FUNCTION_BLOCK C_HTTP_HEADER EXTENDS C_HTTP_BASE
VAR_INPUT
END_VAR
VAR_OUTPUT
END_VAR
VAR
	_FieldName 	: STRING(255);
	_HeaderField: STRING(255);
END_VAR

METHOD Equals : BOOL
VAR_INPUT
	IN_HEADER : POINTER TO C_HTTP_HEADER;
END_VAR
VAR
	_stringInternal 	: STRING(255);
	_stringInput 		: STRING(255);
	_lenString			: INT;
	_i 					: DINT;
END_VAR
IF LEN(IN_HEADER^.Field_Name) <> LEN(THIS^.Field_Name) THEN
	Equals := FALSE;
ELSIF LEN(IN_HEADER^.Header_Field) <> LEN(THIS^.Header_Field) THEN
	Equals := FALSE;
ELSE
	_stringInternal := THIS^.Field_Name;
	_stringInput := IN_HEADER^.Field_Name;
	_lenString := LEN(_stringInternal);
	_i := MEMCMP(ADR(_stringinternal),ADR(_stringInput), _lenString);
	IF _i <> 0 THEN
		Equals := FALSE;
	ELSE
		_stringInternal := THIS^.Header_Field;
		_stringInput := IN_HEADER^.Header_Field;
		_lenString := LEN(_stringInternal);
		_i := MEMCMP(ADR(_stringinternal),ADR(_stringInput), _lenString);
		IF _i <> 0 THEN
			Equals := FALSE;
		ELSE
			Equals := TRUE;
		END_IF
	END_IF
END_IF
END_METHOD

METHOD FB_init : BOOL
VAR_INPUT
	bInitRetains : BOOL; // if TRUE, the retain variables are initialized (warm start / cold start)
	bInCopyCode : BOOL;  // if TRUE, the instance afterwards gets moved into the copy code (online change)
	Name : STRING(255);
END_VAR
_FieldName := Name;
END_METHOD

PROPERTY Field_Name : STRING(255)
GET
Field_Name := _FieldName;
END_GET
SET
_FieldName := Field_Name;
END_SET
END_PROPERTY

PROPERTY Header_Field : STRING(255)
GET
Header_Field := _HeaderField;
END_GET
SET
_HeaderField := Header_Field;
END_SET
END_PROPERTY

METHOD Parse : RETURN_CODE
VAR_INPUT
	IN_STRING	: STRING(255);
END_VAR
VAR 
	_DELIMIT_POSITION : INT;
	_ENDLINE_POSITION : INT;
END_VAR
_DELIMIT_POSITION := FIND(IN_STRING, SUPER^.Header_Delimiter);
IF _DELIMIT_POSITION = 0 THEN
	Parse := ph_lv0.LV0_RETURNCODE.RETURN_ERROR + 1;
ELSE
	_ENDLINE_POSITION := FIND(IN_STRING, SUPER^.Line_Terminator);
	IF _ENDLINE_POSITION = 0 THEN
		Parse := ph_lv0.LV0_RETURNCODE.RETURN_ERROR + 2;
	ELSE
		_FieldName := MID(IN_STRING, _DELIMIT_POSITION - 1, 1);
		_HeaderField := MID(IN_STRING, _ENDLINE_POSITION - (_DELIMIT_POSITION + 2), _DELIMIT_POSITION + 2); 
		Parse := ph_lv0.LV0_RETURNCODE.RETURN_SUCCESS;
	END_IF
END_IF
END_METHOD

METHOD ToString : String(255)
VAR_INPUT
END_VAR
ToString := CONCAT(THIS^.Field_Name,
				CONCAT(SUPER^.Header_Delimiter, 
					CONCAT(THIS^.Header_Field,
						SUPER^.Line_Terminator
					)
				)
			);
END_METHOD

END_FUNCTION_BLOCK

(* stored: Version 1.1.0.1, ProductVersion 3.1.4019.2
   POU C_HTTP_HEADER: Id {f4916d40-e672-4a39-af07-e680b56b31a1}, SpecialFunc None
   Folder Methods: Id {db0984ec-abb7-47f0-9af2-a9a0dd131973}
   Folder Properties: Id {f10153ac-78e0-47cd-a140-91303f7d4cce}
   Method Equals: Id {3902d8e9-12a8-4da2-98b3-710cc8dffbd1}
   Method FB_init: Id {8a629b36-7f23-4909-b667-670fcd0ea299}
   Property Field_Name: Id {04e727c1-324e-4b1d-a850-04650181a981}
   Get Get: Id {503fe4c5-a6d4-4ccd-a58a-24c85418e26c}
   Set Set: Id {ff02c1c9-7548-4158-92cd-b16d33b8e149}
   Property Header_Field: Id {7d96352a-9bf1-4568-85d2-79e6fda2086a}
   Get Get: Id {e60e0c26-7033-4328-845b-f99397daab4c}
   Set Set: Id {794e1deb-29f2-45bf-86d4-91a33d3f7065}
   Method Parse: Id {1a154c0f-ddf2-4163-9ad1-6377946be8c4}
   Method ToString: Id {78ebe571-63bd-4d42-9d18-e745e34f13a3} *)
